FUNCTION_BLOCK A25 EXTENDS GenericSubarea

SUPER^();

METHOD PROTECTED callHardware : BOOL
VAR_INPUT
END_VAR
END_METHOD

METHOD PROTECTED runModules : BOOL
VAR_INPUT
END_VAR
// NETWORK 1
END_METHOD

METHOD PROTECTED setupHardware : BOOL
VAR
	i : INT;
END_VAR
END_METHOD

END_FUNCTION_BLOCK

(* stored: Version 1.1.0.1, ProductVersion 3.1.4024.11
   POU A25: Id {3b04d2e6-0b6c-4c36-b7dd-d9e45e2be25d}, SpecialFunc None
   Method callHardware: Id {3515a28f-6599-4aad-963a-ab704995425b}
   Method runModules: Id {13276b52-bf27-4a0b-a031-31e2c6120e0c}
   Method setupHardware: Id {c528889d-6dba-45a0-ba04-14129789a879} *)
